// SIMATIC S7-200 project (STEP 7-Micro/WIN), CPU 221 REL 01.10

SYMBOL_TABLE USER1
ONN              I0.0
OFF              I0.1
CB_VAO           I0.2
CB_RA            I0.3
XANH             Q0.0
DO               Q0.1
END_SYMBOL_TABLE

ORGANIZATION_BLOCK MAIN:OB1
TITLE=bai tap bai giu xe su dung bo dem couter va lenh so sanh
BEGIN
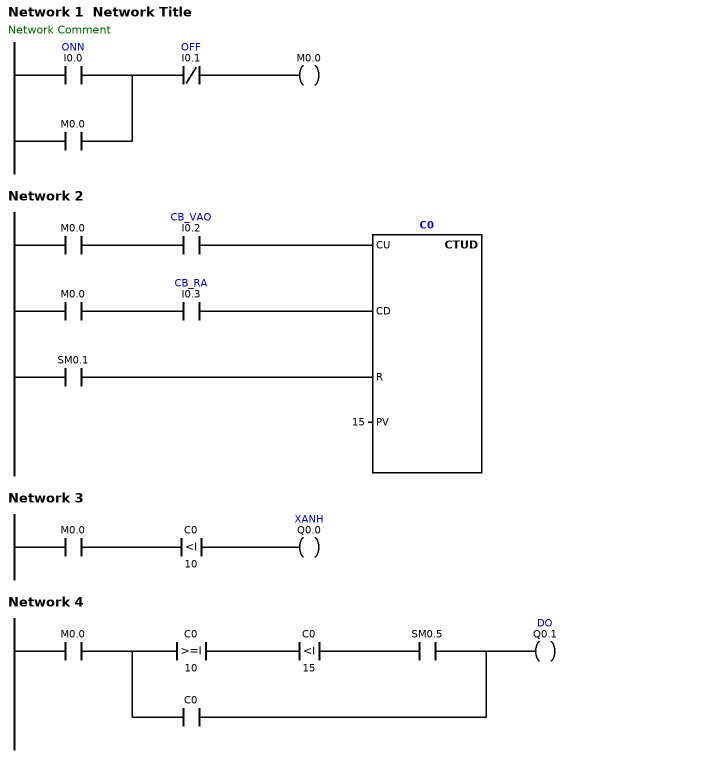
Network 1 // Network Title
// Network Comment
LD     ONN:I0.0
O      M0.0
AN     OFF:I0.1
=      M0.0
Network 2
LD     M0.0
A      CB_VAO:I0.2
LD     M0.0
A      CB_RA:I0.3
LD     SM0.1
CTUD   C0, 15
Network 3
LD     M0.0
AW<    C0, 10
=      XANH:Q0.0
Network 4
LD     M0.0
LDW>=  C0, 10
AW<    C0, 15
A      SM0.5
O      C0
ALD
=      DO:Q0.1
END_ORGANIZATION_BLOCK
